// TIA Portal V17 export
// export: Created 2024-09-02T12:50:29.3054007Z, ExportSetting WithDefaults, DisplayName Totally Integrated Automation Portal, DisplayVersion V17, DisplayName TIA Portal Openness, DisplayVersion V17, DisplayName TIA Portal Version Control Interface, DisplayVersion V17, DisplayName STEP 7 Professional, DisplayVersion V17, DisplayName STEP 7 Safety, DisplayVersion V17, DisplayName WinCC Professional, DisplayVersion V17
TYPE "TypeDirektstarter_in"
// stored: IsFailsafeCompliant false
   STRUCT
      Ready : Bool;   // Bereit (Automatik) / Ready (Automatic)
      MotorON : Bool;   // Motor Ein / Motor On
      SummaryFault : Bool;   // Sammelfehler (Kurzschluss/Überlast) / Group error (short-circuit/overload)
      SummaryWarning : Bool;   // Sammelwarnung / General warning
      Input1 : Bool;   // Eingang 1 / Input 1
      Input2 : Bool;   // Eingang 2 / Input 2
      Input3 : Bool;   // Eingang 3 / Input 3
      Input4 : Bool;   // Eingang 4 / Input 4
      MotorCurrentBit0 : Bool;   // Motorstrom Bit 0 / Motor current Bit 0
      MotorCurrentBit1 : Bool;   // Motorstrom Bit 1 / Motor current Bit 1
      MotorCurrentBit2 : Bool;   // Motorstrom Bit 2 / Motor current Bit 2
      MotorCurrentBit3 : Bool;   // Motorstrom Bit 3 / Motor current Bit 3
      MotorCurrentBit4 : Bool;   // Motorstrom Bit 4 / Motor current Bit 4
      MotorCurrentBit5 : Bool;   // Motorstrom Bit 5 / Motor current Bit 5
      HandModeActive : Bool;   // Betriebsart Hand-Vor-Ort / Manual operating mode - on-site
      RampMode : Bool;   // Rampenbetrieb (OPTION) / Ramp operation (OPTION)
   END_STRUCT;
END_TYPE
